{attribute addProperty BoxType "EP3182-1002-0017"}
{attribute addProperty Id "AI_Standard_ChannelAT %I*ARRAY[0..1] OF AI_Standard_Channel_5763EEB96480DO_OutputsAT %Q*DO_Outputs_E89552221620WcStateAT %I*WcState_F855686C1620InfoDataAT %I*InfoData_BC63D37F80100"}
{attribute addProperty CRC "2212506414"}
{attribute addProperty SizeInBites "176"}
{attribute addProperty SizeInBytes "22"}
TYPE EP3182_E7AA79FE :
STRUCT
	{attribute addProperty Name "AI_Standard_Channel"}
	AI_Standard_Channel : ARRAY[0..1] OF AI_Standard_Channel_5763EEB9;
	{attribute addProperty Name "DO_Outputs"}
	DO_Outputs : DO_Outputs_E8955222;
	{attribute addProperty Name "WcState"}
	WcState : WcState_F855686C;
	{attribute addProperty Name "InfoData"}
	InfoData : InfoData_BC63D37F;
END_STRUCT
END_TYPE

(* stored: Version 1.2.0.0, ProductVersion 3.1.4024.9
   DUT EP3182_E7AA79FE: Id {7c399e1d-4dbd-4409-a676-634aca05ca49} *)
